PROGRAM MAIN
VAR
	counter_x : INT := 0;
	
	test_gcc : FB_MKS422;
	test_vgc : FB_VGC;
	
	ads_watch_dog : FB_ADS_WATCHDOG;
END_VAR

// A counter to confirm that the program is running
counter_x := counter_x + 1;


//test_gcc();
//test_vgc();


ads_watch_dog(
	sNetId := '172.21.148.145.1.1',
	nPort := 851,
	sVarName := 'ADS_connection_counter',
);

END_PROGRAM

(* stored: Version 1.1.0.1, ProductVersion 3.1.4024.2
   POU MAIN: Id {01182312-da8c-444b-9322-7734ec958f62}, SpecialFunc None *)
